Staubli VAL3: GenericPage.pjx

--- GenericPage.pjx ---
Parameters version=s7.6 stackSize=5000 millimeterUnit=true
Program file=getErrorMessage.pgx
Program file=init.pgx
Program file=listFilling.pgx
Program file=readMe.pgx
Program file=start.pgx
Program file=stop.pgx
Data file=GenericPage.dtx
Library alias=ut path=Disk://Tracking/Tools/util/util.pjx

--- GenericPage.dtx ---
num nCOLMAX = 39
num nCOLMIN
public num nColumn
public num nFocused
public num nListSize
num nROWMAX = 12
num nROWMIN
public num nRow
string sErrorMessage
string sErrorMsg[10]
  [0] = "An error has been detected in the Page library *\../*"
  [2] = "Variable sTxtBoxLen[*] has an illegal value"
  [3] = "Variable sTxtBoxPos[*] has an illegal value"
public string sFALSE = "FALSE"
public string sLabel = "-This is a label"
public string sLabelPos = "0;0"
public string sMenu = "F1 F2 ; F4 F5 F6 ; F8"
public string sTRUE = "TRUE"
public string sTitle = "custom EntryBox"
public string sTxtBoxAuthord[3] = "0123456789.-"
public string sTxtBoxCaption[3]
  [0] = "Numeric :"
  [1] = "Boolean :"
  [2] = "List    :"
public string sTxtBoxLen[3]
  [0] = "7"
  [1] = "7"
  [2] = "7"
public string sTxtBoxPos[3]
  [0] = "0;1"
  [1] = "0;2"
  [2] = "0;3"
public string sTxtBoxRange[3] = "-100;100"
public string sTxtBoxType[3]
  [0] = "N"
  [1] = "B"
  [2] = "L6;17;8;5"
public string sTxtBoxVal[3]
  [0] = "421"
  [2] = "0"
public string sListItem0

--- start.pgx ---
program start()
  local string tt[8]
  local num l_nError
begin

  call init(l_nError)

  if l_nError<0

    popUpMsg(sErrorMessage)

  endIf

  //call _str2Array("A;   ; NON",";",tt)

end

--- listFilling.pgx ---
public program listFilling(num x_nListNumber, string& x_sItemList[], num& x_nError)
  local num l_nI
begin

  // This program fills a list object with items

  //

  // Input Param

  //  x_nListNumber  : list number to fill

  //  x_sItemList    : Items to push into the List object

  //

  // Output Param

  //  x_Error : Error code

  //          = 3    : Variable sListItemX doesn't exist

  //

  //--------------------------------------------------------------

  //

  x_nError=0

  switch x_nListNumber

    case 0

      resize(sListItem0,1,size(x_sItemList))

      for l_nI=0 to size(x_sItemList)-1

        sListItem0[l_nI]=x_sItemList[l_nI]

      endFor

    break

    default

      x_nError=3

    break

  endSwitch

  //

end
